SUBAPPLICATION Uebung_020f2 (* DigitalInput_I1 auf DigitalOutput_Q1; FB_TP; Impulsformend *)
  (* Standard: 61499-2; Description: Copyright (c) 2023 Meisterschulen am Ostbahnhof This program and the accompanying materials are made available under the terms of the Eclipse Public License 2.0 which is available at https://www.eclipse.org/legal/epl-2.0/ SPDX-License-Identifier: EPL-2.0 *)
  (* Version 1.0, 2023-10-23, Franz Höpfinger, Meisterschulen am Ostbahnhof *)
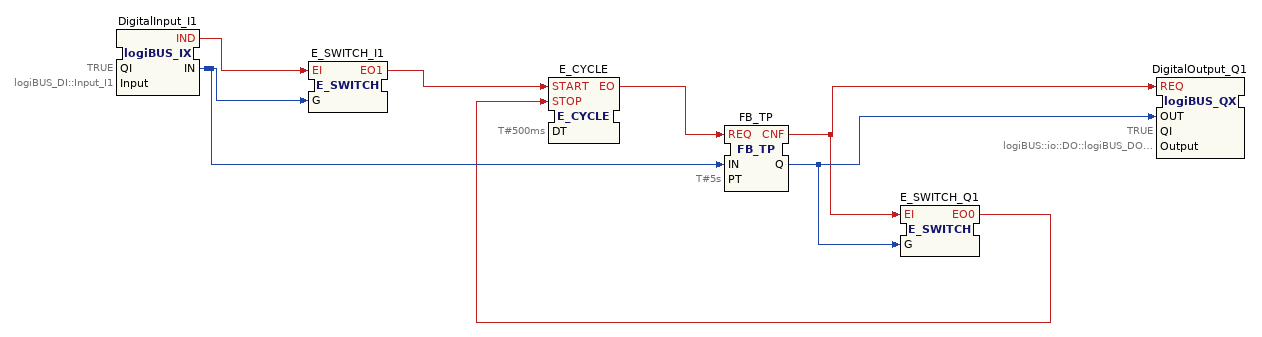
  (* E_CYCLE bestimmt, wie oft FB_TP den ET aktualisert *)
  FBS
    E_SWITCH_I1 : E_SWITCH;
    E_SWITCH_Q1 : E_SWITCH;
    DigitalInput_I1 : logiBUS_IX(QI := TRUE, Input := logiBUS_DI::Input_I1);
    FB_TP : FB_TP(PT := T#5s);
    DigitalOutput_Q1 : logiBUS_QX(QI := TRUE, Output := logiBUS::io::DO::logiBUS_DO::Output_Q1);
    E_CYCLE : E_CYCLE(DT := T#500ms);
  END_FBS
  EVENT_CONNECTIONS
    E_CYCLE.EO TO FB_TP.REQ;
    DigitalInput_I1.IND TO E_SWITCH_I1.EI;
    FB_TP.CNF TO E_SWITCH_Q1.EI;
    E_SWITCH_I1.EO1 TO E_CYCLE.START;
    E_SWITCH_Q1.EO0 TO E_CYCLE.STOP;
    FB_TP.CNF TO DigitalOutput_Q1.REQ;
  END_CONNECTIONS
  DATA_CONNECTIONS
    DigitalInput_I1.IN TO E_SWITCH_I1.G;
    DigitalInput_I1.IN TO FB_TP.IN;
    FB_TP.Q TO DigitalOutput_Q1.OUT;
    FB_TP.Q TO E_SWITCH_Q1.G;
  END_CONNECTIONS
END_SUBAPPLICATION
